{attribute addProperty BoxType "KL2018-0020"}
{attribute addProperty Id "Channel_1Channel_E75BD82E00Channel_2Channel_E75BD82E00Channel_3Channel_E75BD82E00Channel_4Channel_E75BD82E00Channel_5Channel_E75BD82E00Channel_6Channel_E75BD82E00Channel_7Channel_E75BD82E00Channel_8Channel_E75BD82E00"}
{attribute addProperty CRC "2062189974"}
{attribute addProperty SizeInBites "0"}
{attribute addProperty SizeInBytes "0"}
TYPE KL_7AEA8596 :
STRUCT
	{attribute addProperty Name "Channel_1"}
	Channel_1 : Channel_E75BD82E;
	{attribute addProperty Name "Channel_2"}
	Channel_2 : Channel_E75BD82E;
	{attribute addProperty Name "Channel_3"}
	Channel_3 : Channel_E75BD82E;
	{attribute addProperty Name "Channel_4"}
	Channel_4 : Channel_E75BD82E;
	{attribute addProperty Name "Channel_5"}
	Channel_5 : Channel_E75BD82E;
	{attribute addProperty Name "Channel_6"}
	Channel_6 : Channel_E75BD82E;
	{attribute addProperty Name "Channel_7"}
	Channel_7 : Channel_E75BD82E;
	{attribute addProperty Name "Channel_8"}
	Channel_8 : Channel_E75BD82E;
END_STRUCT
END_TYPE

(* stored: Version 1.2.0.0, ProductVersion 3.1.4024.9
   DUT KL_7AEA8596: Id {0366f5d2-4b40-4656-b82e-4747e338331b} *)
